// TIA Portal V21 export
VAR_GLOBAL   // PLC tag table "ClusterSendDigitali"
END_VAR
VAR_GLOBAL CONSTANT   // user constants
   K_SegnaleVersoCluster_Consenso : Int := 1;
END_VAR
